// SIMATIC S7-200 project (STEP 7-Micro/WIN), CPU 224XP REL 02.01

SYMBOL_TABLE USUARIO1
ASCENDENTE       I0.0
DESCENDENTE      I0.1
RESET            I0.2
display          MB10
contador         MW0
END_SYMBOL_TABLE

SYMBOL_TABLE Símbolos S7-200
Siempre_ON       SM0.0    // Siempre ON
Primer_ciclo_ON  SM0.1    // ON sólo en el primer ciclo
Reloj_1s         SM0.5    // Reloj ON durante 0,5 s, OFF durante 0,5 s, tiempo de ciclo = 1 s.
END_SYMBOL_TABLE

ORGANIZATION_BLOCK PRINCIPAL:OB1
TITLE=COMENTARIOS DEL PROGRAMA
BEGIN
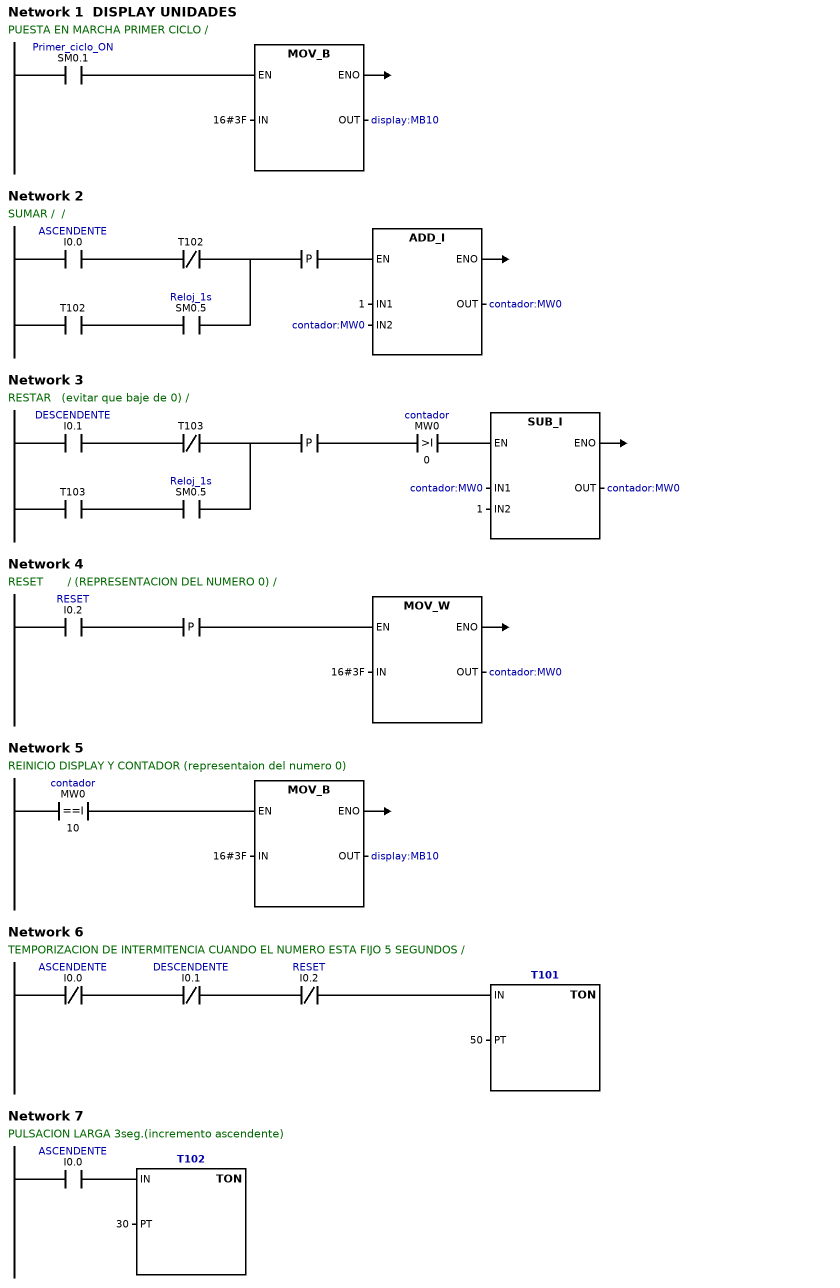
Network 1 // DISPLAY UNIDADES


// PUESTA EN MARCHA PRIMER CICLO
// 
LD     Primer_ciclo_ON:SM0.1
MOVB   16#3F, display:MB10
Network 2
// SUMAR
// 
// 
// (network saved uncompiled; LAD cells follow)
// row 0: c0 -| |- ASCENDENTE:I0.0  c1 -|/|- T102 v  c2 -|P|-  c3 [ADD_I EN:=power@row0, IN1:=1, IN2:=contador:MW0, ENO=>power, OUT=>contador:MW0]  c4 ->
// row 1: c0 -| |- T102  c1 -| |- Reloj_1s:SM0.5 ^  c3 [box]
Network 3
// RESTAR   (evitar que baje de 0)
// 
// (network saved uncompiled; LAD cells follow)
// row 0: c0 -| |- DESCENDENTE:I0.1  c1 -|/|- T103 v  c2 -|P|-  c3 -|>I|- contador:MW0, 0  c4 [SUB_I EN:=power@row0, IN1:=contador:MW0, IN2:=1, ENO=>power, OUT=>contador:MW0]  c5 ->
// row 1: c0 -| |- T103  c1 -| |- Reloj_1s:SM0.5 ^  c4 [box]
Network 4
// RESET      
// (REPRESENTACION DEL NUMERO 0)
// 
LD     RESET:I0.2
EU
MOVW   16#3F, contador:MW0
Network 5
// REINICIO DISPLAY Y CONTADOR (representaion del numero 0)
LDW=   contador:MW0, 10
MOVB   16#3F, display:MB10
Network 6
// TEMPORIZACION DE INTERMITENCIA CUANDO EL NUMERO ESTA FIJO 5 SEGUNDOS
// 
LDN    ASCENDENTE:I0.0
AN     DESCENDENTE:I0.1
AN     RESET:I0.2
TON    T101, 50
Network 7
// PULSACION LARGA 3seg.(incremento ascendente)
// (network saved uncompiled; LAD cells follow)
// row 0: c0 -| |- ASCENDENTE:I0.0  c1 [TON T102 IN:=power@row0, PT:=30]
// row 1: c1 [box]
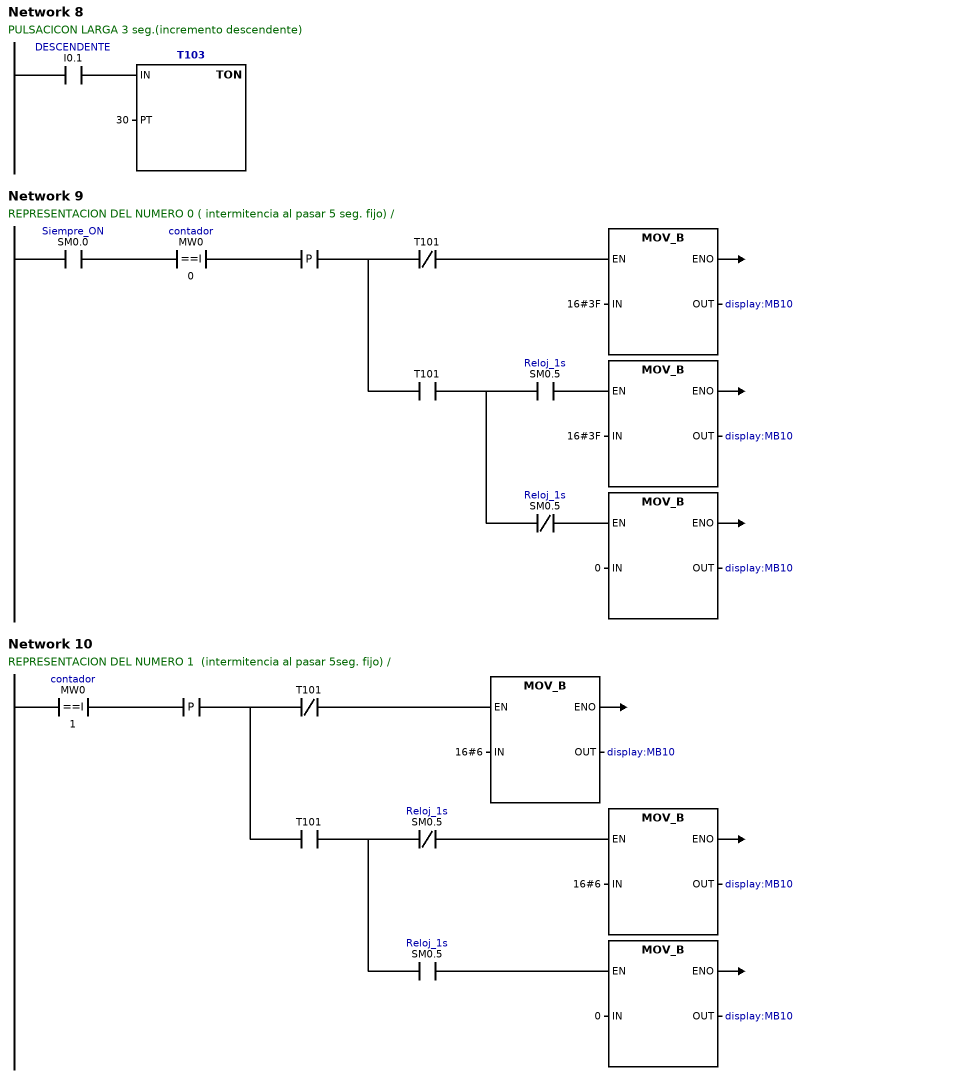
Network 8
// PULSACICON LARGA 3 seg.(incremento descendente)
// (network saved uncompiled; LAD cells follow)
// row 0: c0 -| |- DESCENDENTE:I0.1  c1 [TON T103 IN:=power@row0, PT:=30]
// row 1: c1 [box]
Network 9
// REPRESENTACION DEL NUMERO 0 ( intermitencia al pasar 5 seg. fijo)
// 
// (network saved uncompiled; LAD cells follow)
// row 0: c0 -| |- Siempre_ON:SM0.0  c1 -|==I|- contador:MW0, 0  c2 -|P|-  v  c3 -|/|- T101  c4 --  c5 [MOV_B EN:=power@row0, IN:=16#3F, ENO=>power, OUT=>display:MB10]  c6 ->
// row 1: c2 ^v  c5 [box]
// row 2: c2 ^  c3 -| |- T101 v  c4 -| |- Reloj_1s:SM0.5  c5 [MOV_B EN:=power@row2, IN:=16#3F, ENO=>power, OUT=>display:MB10]  c6 ->
// row 3: c3 ^v  c5 [box]
// row 4: c3 ^  c4 -|/|- Reloj_1s:SM0.5  c5 [MOV_B EN:=power@row4, IN:=0, ENO=>power, OUT=>display:MB10]  c6 ->
// row 5: c5 [box]
Network 10
// REPRESENTACION DEL NUMERO 1  (intermitencia al pasar 5seg. fijo)
// 
LDW=   contador:MW0, 1
EU
LPS
AN     T101
MOVB   16#6, display:MB10
LPP
A      T101
LPS
AN     Reloj_1s:SM0.5
MOVB   16#6, display:MB10
LPP
A      Reloj_1s:SM0.5
MOVB   0, display:MB10
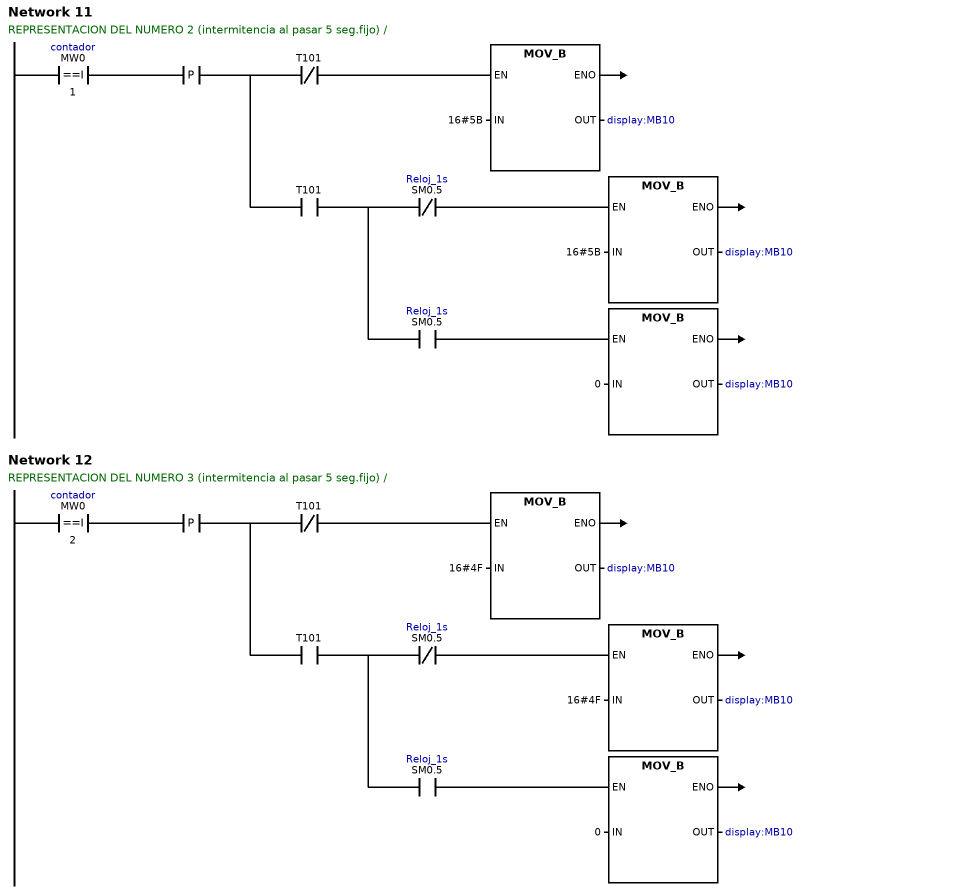
Network 11
// REPRESENTACION DEL NUMERO 2 (intermitencia al pasar 5 seg.fijo)
// 
LDW=   contador:MW0, 1
EU
LPS
AN     T101
MOVB   16#5B, display:MB10
LPP
A      T101
LPS
AN     Reloj_1s:SM0.5
MOVB   16#5B, display:MB10
LPP
A      Reloj_1s:SM0.5
MOVB   0, display:MB10
Network 12
// REPRESENTACION DEL NUMERO 3 (intermitencia al pasar 5 seg.fijo)
// 
LDW=   contador:MW0, 2
EU
LPS
AN     T101
MOVB   16#4F, display:MB10
LPP
A      T101
LPS
AN     Reloj_1s:SM0.5
MOVB   16#4F, display:MB10
LPP
A      Reloj_1s:SM0.5
MOVB   0, display:MB10
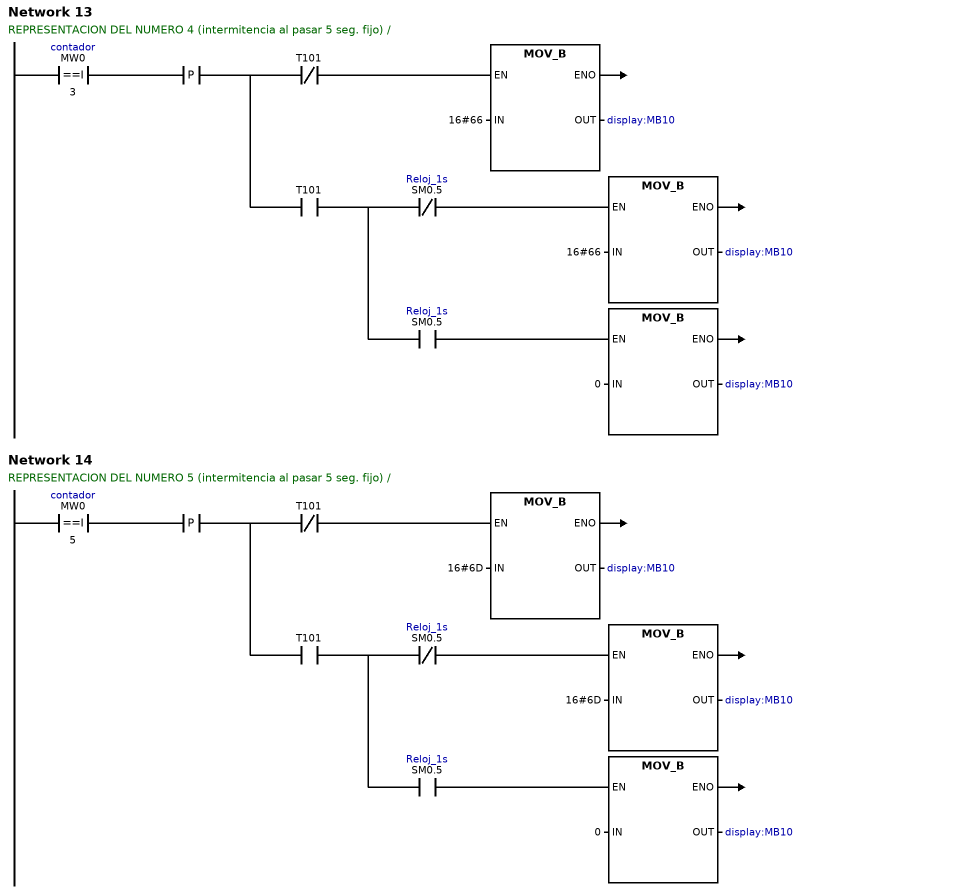
Network 13
// REPRESENTACION DEL NUMERO 4 (intermitencia al pasar 5 seg. fijo)
// 
LDW=   contador:MW0, 3
EU
LPS
AN     T101
MOVB   16#66, display:MB10
LPP
A      T101
LPS
AN     Reloj_1s:SM0.5
MOVB   16#66, display:MB10
LPP
A      Reloj_1s:SM0.5
MOVB   0, display:MB10
Network 14
// REPRESENTACION DEL NUMERO 5 (intermitencia al pasar 5 seg. fijo)
// 
LDW=   contador:MW0, 5
EU
LPS
AN     T101
MOVB   16#6D, display:MB10
LPP
A      T101
LPS
AN     Reloj_1s:SM0.5
MOVB   16#6D, display:MB10
LPP
A      Reloj_1s:SM0.5
MOVB   0, display:MB10
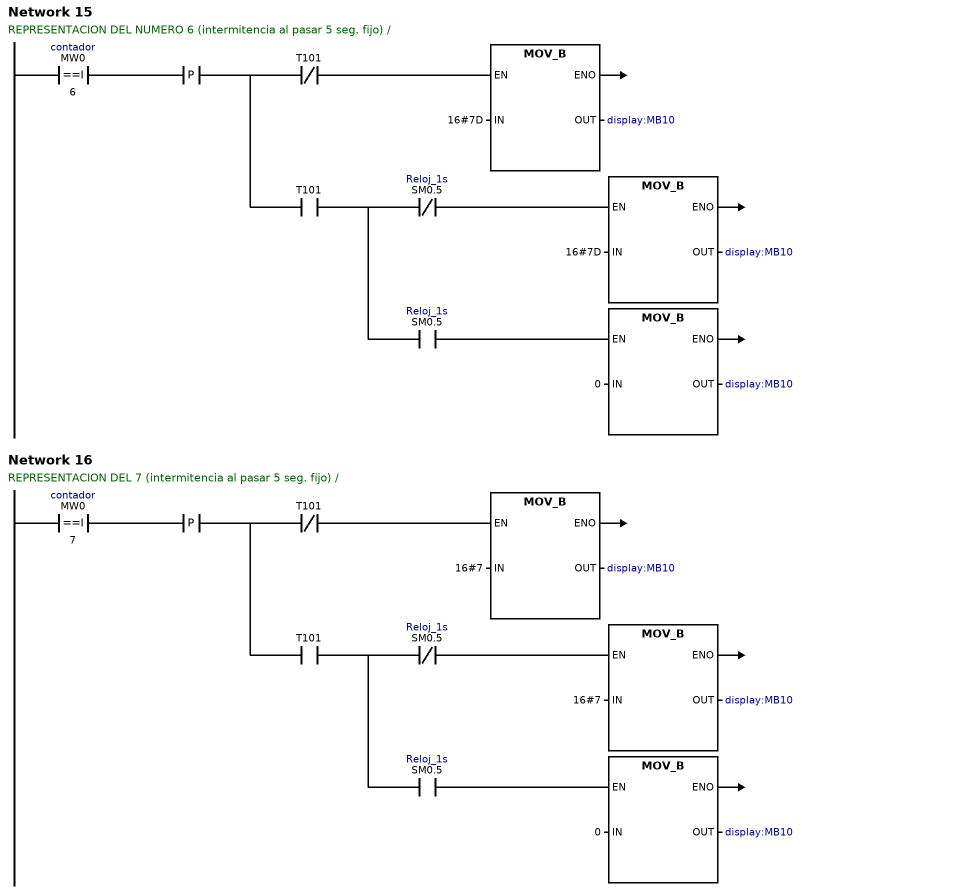
Network 15
// REPRESENTACION DEL NUMERO 6 (intermitencia al pasar 5 seg. fijo)
// 
LDW=   contador:MW0, 6
EU
LPS
AN     T101
MOVB   16#7D, display:MB10
LPP
A      T101
LPS
AN     Reloj_1s:SM0.5
MOVB   16#7D, display:MB10
LPP
A      Reloj_1s:SM0.5
MOVB   0, display:MB10
Network 16
// REPRESENTACION DEL 7 (intermitencia al pasar 5 seg. fijo)
// 
LDW=   contador:MW0, 7
EU
LPS
AN     T101
MOVB   16#7, display:MB10
LPP
A      T101
LPS
AN     Reloj_1s:SM0.5
MOVB   16#7, display:MB10
LPP
A      Reloj_1s:SM0.5
MOVB   0, display:MB10
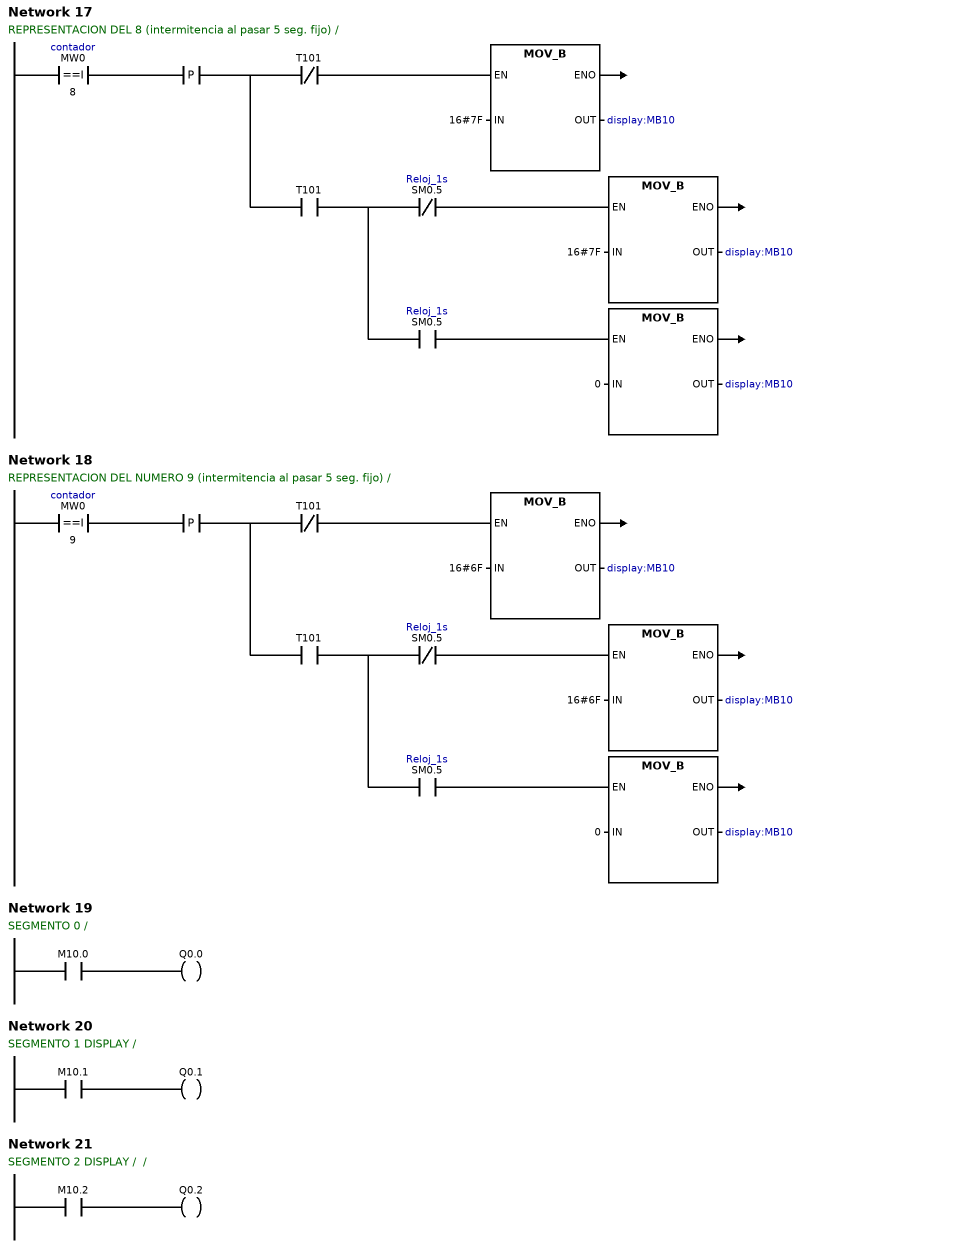
Network 17
// REPRESENTACION DEL 8 (intermitencia al pasar 5 seg. fijo)
// 
LDW=   contador:MW0, 8
EU
LPS
AN     T101
MOVB   16#7F, display:MB10
LPP
A      T101
LPS
AN     Reloj_1s:SM0.5
MOVB   16#7F, display:MB10
LPP
A      Reloj_1s:SM0.5
MOVB   0, display:MB10
Network 18
// REPRESENTACION DEL NUMERO 9 (intermitencia al pasar 5 seg. fijo)
// 
LDW=   contador:MW0, 9
EU
LPS
AN     T101
MOVB   16#6F, display:MB10
LPP
A      T101
LPS
AN     Reloj_1s:SM0.5
MOVB   16#6F, display:MB10
LPP
A      Reloj_1s:SM0.5
MOVB   0, display:MB10
Network 19
// SEGMENTO 0
// 
LD     M10.0
=      Q0.0
Network 20
// SEGMENTO 1 DISPLAY
// 
LD     M10.1
=      Q0.1
Network 21
// SEGMENTO 2 DISPLAY
// 
// 
LD     M10.2
=      Q0.2
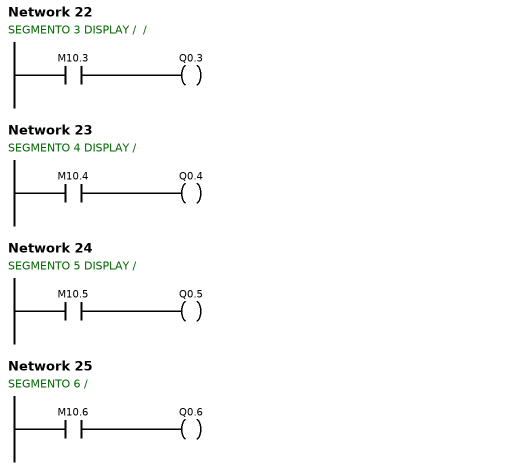
Network 22
// SEGMENTO 3 DISPLAY
// 
// 
LD     M10.3
=      Q0.3
Network 23
// SEGMENTO 4 DISPLAY
// 
LD     M10.4
=      Q0.4
Network 24
// SEGMENTO 5 DISPLAY
// 
LD     M10.5
=      Q0.5
Network 25
// SEGMENTO 6
// 
LD     M10.6
=      Q0.6
END_ORGANIZATION_BLOCK
